Staubli VAL3: DealRobMaster.pjx

--- DealRobMaster.pjx ---
Parameters version=s7.8.3 stackSize=5000 millimeterUnit=true
Program file=chkIsFileExsit.pgx
Program file=Init.pgx
Program file=JudgePeak.pgx
Program file=Main.pgx
Program file=MainKey.pgx
Program file=OnePathConvert.pgx
Program file=OnF1.pgx
Program file=OnF2.pgx
Program file=OnF3.pgx
Program file=OnF4.pgx
Program file=OnF5.pgx
Program file=OnF6.pgx
Program file=OnF7.pgx
Program file=OnF8.pgx
Program file=readFileList.pgx
Program file=Refresh.pgx
Program file=RefreshList.pgx
Program file=selectFile.pgx
Program file=start.pgx
Program file=stop.pgx
Data file=DealRobMaster.dtx
Library alias=master path=Disk://template/robotmaster/robotmaster.pjx
Library alias=user path=Disk://userPage/USERPAGE.pjx
Library alias=prd path=Disk://template/normalPath/normalPath.pjx
Library alias=Frame path=Disk://Frame/Frame.pjx

--- DealRobMaster.dtx ---
mdesc mNomSpeed
public string sFileList
public string sDeli[4]
  [0] = "A"
  [1] = "C"
  [2] = "B"
  [3] = "D"
bool bUserRefresh
bool bListRefresh
bool bExit
num nSelected
string sItem
string sFolder = "Disk://robmaster/"
string sOutputFolder = "Disk://Traj/"
string sFileTemp
frame fFrame = {fatherId=world[0]}
tool tTool = {fatherId=flange[0], ioLink=valve1}

--- Main.pgx ---
program Main()
  local num l_nKey
begin
  //
 do
    call Refresh()
    call RefreshList()
    call user:setList("路径",sFileList,bUserRefresh,bListRefresh,nSelected,sItem,l_nKey)
    bUserRefresh=false
    bListRefresh=false
    call MainKey(l_nKey)
    delay(0)
  until bExit

end

--- chkIsFileExsit.pgx ---
program chkIsFileExsit(string x_sFileName, string x_sTargetFolder, bool& x_bRes)
  local num l_ni
begin
  //检查文件x_sFileName在目标文件夹中x_sTargetFolder是否存在
  x_bRes=false
  resize(sFileTemp,1,1)
  sFileTemp[0]=""
  if (libList(x_sTargetFolder,sFileTemp)==false)
    return
  endIf
  //
  for l_ni=0 to size(sFileTemp)-1
    if x_sFileName==sFileTemp[l_ni]
      x_bRes=true
      return
    endIf
  endFor

end

--- Init.pgx ---
program Init()
  local num l_ni
begin

  bUserRefresh=bListRefresh=true
  //
  bExit=false
  //
  call readFileList(sFolder,sFileList)
  //call selectFile(sDeli,sFileList)
end

--- JudgePeak.pgx ---
program JudgePeak()
begin
  //判断路径中的转折点
  //
end

--- MainKey.pgx ---
program MainKey(num x_nKey)
  local num l_nKey
begin
  switch x_nKey
    //
    case 271
      call OnF1()
    break
    //
    case 272
      call OnF2()
    break
    //
    case 273
      call OnF3()
    break
    //
    case 274
      call OnF4()
    break
    //
    case 275
    break
    //
    case 276
      call OnF6()
    break
    //save
    case 277
      call OnF7()
    break
    //返回
    case 278,255
      call OnF8("是否返回?")
    break
  endSwitch
end

--- OnePathConvert.pgx ---
program OnePathConvert(string x_sFolder, string x_sMasterFile, string x_sOutputFolder, bool& x_bRes)
  local num l_nsize
  local num l_ni
  local num l_nj
  local joint l_jJoint[2]
begin
  //载入master文件
  x_bRes=false

  if master:libLoad(x_sFolder+x_sMasterFile)!=0
    return
  endIf
  //由于mastercam生成出来的真实坐标位置是保存在tTool里的。
  prd:fFrmMaster.trsf=master:fUserFrame.trsf
  Frame:fFrame["Frame1"].trsf=master:fUserFrame.trsf
  prd:tTool.trsf=master:tTool.trsf
  prd:sFrameName=""
  prd:sToolName=""
  //补偿量(mm)
  prd:nCompDelta=0.002
  //取个数
  l_nsize=size(master:ptRoutingPath)
  //存个数
  resize(prd:pDemo,1,l_nsize)
  resize(prd:sPtParameter,1,l_nsize)
  for l_ni=0 to l_nsize-1
    prd:sPtParameter[l_ni]="-1/-1/-1/-1/-1/-1"
  endFor
  //
  prd:mNormal=master:mdLineBlend
  prd:mJoint=master:mdJointBlend
  prd:mJoint.vel=100
  prd:mJoint.accel=prd:mJoint.decel=50
  prd:mJoint.tvel=300
  prd:mJoint.reach=prd:mJoint.leave=1
  //
  l_nj=0
  for l_ni=0 to l_nsize-1
    //点复制
    prd:pDemo[l_ni].trsf=master:ptRoutingPath[l_ni].trsf
    prd:pDemo[l_ni].config.shoulder=ssame
    prd:pDemo[l_ni].config.elbow=esame
    prd:pDemo[l_ni].config.wrist=wsame
    //
    if l_ni!=0
      if (pointToJoint(master:tTool,master:jtPark,master:ptRoutingPath[l_ni],l_jJoint[1])==false)
        popUpMsg("转换失败："+toString("",l_ni))
        return
      endIf
      if(pointToJoint(master:tTool,master:jtPark,master:ptRoutingPath[l_ni-1],l_jJoint[0])==false)
        popUpMsg("转换失败："+toString("",l_ni-1))
        return
      endIf
      //如果超出50，则把l_ni的数据赋值到nPeak[l_nj]
      if abs(l_jJoint[1].j6-l_jJoint[0].j6)>50
        prd:nPeak[l_nj]=l_ni
        l_nj=l_nj+1
        insert(prd:nPeak[l_nj])
      endIf
    endIf
  endFor
  delete(prd:nPeak[l_nj])
  //保存程序
  prd:libSave(x_sOutputFolder+x_sMasterFile)
  Frame:libSave()
  x_bRes=true
end

--- OnF1.pgx ---
program OnF1()
  local bool l_bRes
  local string l_sYesNo[2]
begin
  //单一路径转化
  //
  //检查文件是否已经存在
  call chkIsFileExsit(sItem,sOutputFolder,l_bRes)
  //存在，询问
  if l_bRes
    l_sYesNo[0]="是"
    l_sYesNo[1]="否"
    call user:yes_no("文件已存在，是否覆盖?",l_sYesNo,l_bRes)
    bUserRefresh=true
    if !l_bRes
      return
    else
      $delete(sOutputFolder+sItem)
    endIf
  endIf
  //

  //转换文件
  call OnePathConvert(sFolder,sItem,sOutputFolder,l_bRes)
  if l_bRes
    popUpMsg("转换完成")
  else
    popUpMsg("文件转换失败!")
  endIf
end

--- OnF2.pgx ---
program OnF2()
  local num l_ni
  local bool l_bRes
begin
  //全部转换
  for l_ni=0 to size(sFileList)-1
    call OnePathConvert(sFolder,sFileList[l_ni],sOutputFolder,l_bRes)
    if !l_bRes
      popUpMsg(sFileList[l_ni]+"文件转换失败!")
      logMsg(sFileList[l_ni]+"文件转换失败!")
      wait(getKey()==278)
    endIf
  endFor
  popUpMsg("转换完成")
end

--- OnF3.pgx ---
program OnF3()
  local string l_sYesNo[2]
  local num l_i
begin
  //删除
  l_sYesNo[0]="是"
  l_sYesNo[1]="否"
  call user:questionDialog("是否删除此路径?",l_sYesNo,l_i)
  if l_i==0 or l_i==1
    if sFileList[nSelected]!=""
      libDelete(sFolder+sFileList[nSelected])
      delete(sFileList[nSelected])
      bListRefresh=true
    endIf
  endIf
  bUserRefresh=true

end

--- OnF4.pgx ---
program OnF4()
begin
end

--- OnF5.pgx ---
program OnF5()
begin
end

--- OnF6.pgx ---
program OnF6()
begin
end

--- OnF7.pgx ---
program OnF7()
begin
  //

end

--- readFileList.pgx ---
public program readFileList(string x_sFileFolder, string& x_sFileList[])
begin
  //读取robotmaster生成的全部文件列表
  resize(x_sFileList,1,1)
  x_sFileList[0]=""
  if !libList(x_sFileFolder,x_sFileList)
    logMsg("读取文件列表错误")
  endIf
end

--- Refresh.pgx ---
program Refresh()
begin
  //
  if bUserRefresh
    cls()
    userPage()
    gotoxy(1,1)
    put("F1->选中路径转换")
    gotoxy(1,13)
    put("转换")
    gotoxy(1,2)
    put("F2->全部转换")
    gotoxy(6,13)
    put("全部")
    gotoxy(1,3)
    put("F3->删除路径")
    gotoxy(11,13)
    put("删除")
//    gotoxy(1,4)
//    put("F4->")
//    gotoxy(16,13)
//    put("")
    //
//    gotoxy(1,6)
//    put("F6->")
//    gotoxy(26,13)
//    put("")
//    gotoxy(1,7)
//    put("F7->")
//    gotoxy(31,13)
//    put("")
    gotoxy(1,7)
    put("F8->返回")
    gotoxy(36,13)
    put("返回")
  endIf
end

--- RefreshList.pgx ---
program RefreshList()
  local num l_ni
begin

end

--- selectFile.pgx ---
public program selectFile(string& x_sDelimiter[], string& x_sList[])
  local num l_ni
  local num l_nj
begin
  //根据x_sDelimiter(分隔符)找出需要的文件
  for l_nj=0 to size(x_sList)-1
    if x_sList[l_nj]!=""
      for l_ni=0 to size(x_sDelimiter)-1
        if left(x_sList[l_nj],1)==x_sDelimiter[l_ni]
          l_ni=size(x_sDelimiter)
        endIf
        if l_ni==size(x_sDelimiter)-1
          delete(x_sList[l_nj])
          l_nj=l_nj-1
        endIf
      endFor
    endIf
  endFor
end
